# EPICS autosave request: iocBoot/iocEnergy_32ID/auto_settings.req
file "energy_settings.req", P=$(P), R=$(R)
file "energy_32ID_settings.req", P=$(P), R=$(R)
